// Mitsubishi GX Works2 project: m07   PLC: Q02/Q02H

PROGRAM MAIN
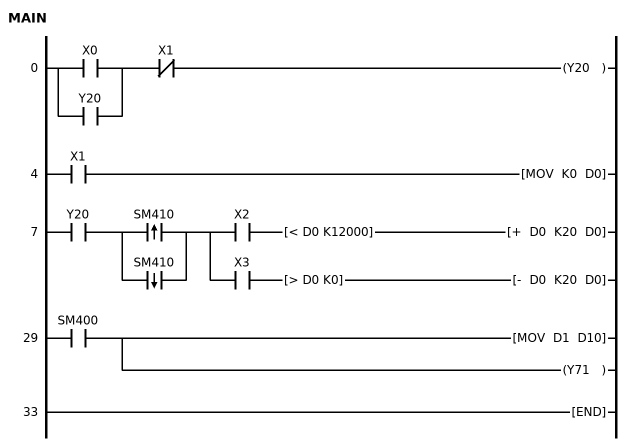
0     LD      X0
      OR      Y20
      ANI     X1
      OUT     Y20
4     LD      X1
      MOV     K0 D0
7     LD      Y20
      LDP     SM410
      ORF     SM410
      ANB
      MPS
      AND     X2
      AND<    D0 K12000
      +       D0 K20 D0
      MPP
      AND     X3
      AND>    D0 K0
      -       D0 K20 D0
29    LD      SM400
      MOV     D1 D10
      OUT     Y71
33    END
END_PROGRAM
